FUNCTION_BLOCK E_RF_TRIG (* Boolean falling and rising edge detection *)
  (* Standard: 61499-1 Annex A; Description: Copyright (c) 2017 fortiss GmbH, HR Agrartechnik GmbH This program and the accompanying materials are made available under the terms of the Eclipse Public License 2.0 which is available at https://www.eclipse.org/legal/epl-2.0/ SPDX-License-Identifier: EPL-2.0 *)
  (* Version 1.0, 2026-05-08, Franz Höpfinger, HR Agrartechnik GmbH, initial API and implementation and/or initial documentation *)
  PACKAGE adapter::events::unidirectional;
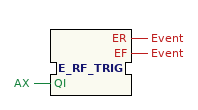
  EVENT_OUTPUT
    ER; (* confirmation that a rising edge was detected *)
    EF; (* confirmation that a falling edge was detected *)
  END_EVENT
  SOCKETS
    QI : adapter::types::unidirectional::AX; (* value to check for a rising or falling edge *)
  END_SOCKETS
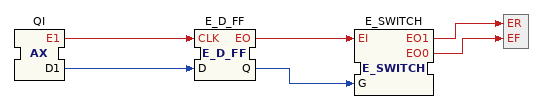
  FBS
    E_D_FF : iec61499::events::E_D_FF;
    E_SWITCH : iec61499::events::E_SWITCH;
  END_FBS
  EVENT_CONNECTIONS
    E_D_FF.EO TO E_SWITCH.EI;
    E_SWITCH.EO1 TO ER;
    E_SWITCH.EO0 TO EF;
    QI.E1 TO E_D_FF.CLK;
  END_CONNECTIONS
  DATA_CONNECTIONS
    E_D_FF.Q TO E_SWITCH.G;
    QI.D1 TO E_D_FF.D;
  END_CONNECTIONS
END_FUNCTION_BLOCK
